Staubli VAL3: GetFirmVersion.pgx

program GetFirmVersion(string& answer)
begin
//*******************************************************************************
//*   ______
//*  / _____) /|
//* | |      / /
//* | | /\  / /
//* | | \ \/ /  _      Copyright (c) KEOLABS, 2016
//* | |  \__/  | |        http://www.keolabs.com
//* | |________| |
//*  \__________/
//*
//********************************************************************************
//*@file          : GetFirmVersion
//*@author        : Yves Ragot
//*@version       : $Id: GetFirmVersion.pgx 1376 2016-11-22 14:02:21Z yves $
//*@brief         : Get firmware version (VAL3 version)
//*
//*******************************************************************************/

   answer = left(getVersion("VAL3"), 20)
//   answer = left(getVersion("Starc"), 20)

end
